// Deklarationsbereich

PROGRAM MAIN
VAR
	bIn1, bIn2, bOut : BOOL;
END_VAR

// Anweisungsbereich

bOut := bIn1 AND bIn2;		//Logisches AND

(*
Comment for multiple lines
*)

END_PROGRAM

(* stored: Version 1.1.0.1, ProductVersion 3.1.4024.12
   POU MAIN: Id {c32b958a-3105-41d9-9190-232c80de93b2}, SpecialFunc None *)
